TYPE sRollerDoor :
STRUCT
	ManualOpenRequest	: BOOL;
	ManualCloseRequest	: BOOL;
	AutoOpenRequest	 	: BOOL;
	AutoCloseRequest	: BOOL;
		
	CommandOpenOutput	AT %Q* : BOOL;		
	CommandCloseOutput	AT %Q* : BOOL;
	
	StatusOpenedInput	AT %I* : BOOL; //This is Normally Closed
	StatusClosedInput	AT %I* : BOOL; //This is Normally Closed
	
	// DOOR_OPEN_SWITCH AT %I*: BOOL;// REAL WORLD SWITCH INPUT
	// DOOR_CLOSED_SWITCH AT %I*: BOOL; // REAL WORLD SWITCH INPUT
	DOOR_CLEAR AT %I* : BOOL; // LIGHT CURTAIN CLEAR
	// RUN_UP AT %Q* : BOOL; // DISCRETE OUTPUT FOR RAISE DOOR COMMAND
	// RUN_DOWN AT %Q* : BOOL; // DISCRETE OUTPUT FOR LOWER DOOR COMMAND
	DOOR_OPEN:BOOL; // DOOR CURRENT POSITION IS OPEN
	DOOR_CLOSED:BOOL; // DOOR CURRENT POSITION IS CLOSED
	OPEN_REQUEST:BOOL; // PLC REQUESTING ROLL DOOR TO OPEN
	CLOSE_REQUEST:BOOL; // PLC REQUESTING ROLL DOOR TO CLOSE
	UP_SWITCH_IS_ON:BOOL; // DOOR SWITCH FOR UP POSITION IS ON
	UP_SWITCH_IS_OFF:BOOL; // DOOR SWITCH FOR UP POSITION IS OFF
	DOWN_SWITCH_IS_ON:BOOL; // DOOR SWITCH FOR DOWN POSITION IS ON
	DOWN_SWITCH_IS_OFF:BOOL; // DOOR SWITCH FOR DOWN POSITION IS OFF
	
	
	DOOR_IS_UP_TimerOn : TON;
	DOOR_IS_UP_TimerOn_Done_Bit: BOOL;
	DOOR_IS_UP_TIMER_ON_ELAPSED : TIME;
	
	DOOR_IS_UP_TimerOFF : TOF;
	DOOR_IS_UP_TimerOFF_Done_Bit: BOOL;
	DOOR_IS_UP_TIMER_OFF_ELAPSED : TIME;
	
	DOOR_IS_DOWN_TimerOn : TON;
	DOOR_IS_DOWN_TimerOn_Done_Bit: BOOL;
	DOOR_IS_DOWN_TIMER_ON_ELAPSED : TIME;
	
	DOOR_IS_DOWN_TimerOFF : TOF;
	DOOR_IS_DOWN_TimerOFF_Done_Bit: BOOL;
	DOOR_IS_DOWN_TIMER_OFF_ELAPSED : TIME;
	
END_STRUCT
END_TYPE

(* stored: Version 1.1.0.1, ProductVersion 3.1.4024.12
   DUT sRollerDoor: Id {10244a97-9bb9-4822-9828-9cd30e168ce4} *)
